# EPICS autosave request: iocBoot/iocFOFB/auto_settings.req
file "FOFB_settings.req",               P=$(P),  R=$(R),  S=$(S)

file "NDPluginBase_settings_mod.req",   P=$(P),  R=$(R)GEN_CH0
file "NDStdArrays_settings.req",        P=$(P),  R=$(R)GEN_CH0
file "NDPluginBase_settings_mod.req",   P=$(P),  R=$(R)GEN_CH1
file "NDStdArrays_settings.req",        P=$(P),  R=$(R)GEN_CH1
file "NDPluginBase_settings_mod.req",   P=$(P),  R=$(R)GEN_CH2
file "NDStdArrays_settings.req",        P=$(P),  R=$(R)GEN_CH2
file "NDPluginBase_settings_mod.req",   P=$(P),  R=$(R)GEN_CH3
file "NDStdArrays_settings.req",        P=$(P),  R=$(R)GEN_CH3
file "NDPluginBase_settings_mod.req",   P=$(P),  R=$(R)GEN_CH4
file "NDStdArrays_settings.req",        P=$(P),  R=$(R)GEN_CH4
file "NDPluginBase_settings_mod.req",   P=$(P),  R=$(R)GEN_CH5
file "NDStdArrays_settings.req",        P=$(P),  R=$(R)GEN_CH5
file "NDPluginBase_settings_mod.req",   P=$(P),  R=$(R)GEN_CH6
file "NDStdArrays_settings.req",        P=$(P),  R=$(R)GEN_CH6
file "NDPluginBase_settings_mod.req",   P=$(P),  R=$(R)GEN_CH7
file "NDStdArrays_settings.req",        P=$(P),  R=$(R)GEN_CH7
file "NDPluginBase_settings_mod.req",   P=$(P),  R=$(R)GEN_CH8
file "NDStdArrays_settings.req",        P=$(P),  R=$(R)GEN_CH8
file "NDPluginBase_settings_mod.req",   P=$(P),  R=$(R)GEN_CH9
file "NDStdArrays_settings.req",        P=$(P),  R=$(R)GEN_CH9
file "NDPluginBase_settings_mod.req",   P=$(P),  R=$(R)GEN_CH10
file "NDStdArrays_settings.req",        P=$(P),  R=$(R)GEN_CH10
file "NDPluginBase_settings_mod.req",   P=$(P),  R=$(R)GEN_CH11
file "NDStdArrays_settings.req",        P=$(P),  R=$(R)GEN_CH11
file "NDPluginBase_settings_mod.req",   P=$(P),  R=$(R)GEN_CH12
file "NDStdArrays_settings.req",        P=$(P),  R=$(R)GEN_CH12
file "NDPluginBase_settings_mod.req",   P=$(P),  R=$(R)GEN_CH13
file "NDStdArrays_settings.req",        P=$(P),  R=$(R)GEN_CH13
file "NDPluginBase_settings_mod.req",   P=$(P),  R=$(R)GEN_CH14
file "NDStdArrays_settings.req",        P=$(P),  R=$(R)GEN_CH14
file "NDPluginBase_settings_mod.req",   P=$(P),  R=$(R)GEN_CH15
file "NDStdArrays_settings.req",        P=$(P),  R=$(R)GEN_CH15
